// TIA Portal V20 export
FUNCTION "CallManualOperationLines_Unit1" : Void   // FC80, LAD
// stored: SetENOAutomatically false
   VAR_TEMP
      StatusEm : Array[0..13] of Struct
         Status : Array[0..40] of Word;
      END_STRUCT;
      errorIDEm : Array[0..13] of Struct
         errorID : Array[0..40] of Word;
      END_STRUCT;
      disableUnit1 : Bool;
      TempAxisCommands : "LBC_typeAxis64PosManualCommands";
      TempAxisMonitoring : "LBC_typeAxis64PosProcessValues";
      TempSoftCam : Array[0..8] of "LER_typeSoftCamParameter";
   END_VAR
   VAR CONSTANT
      MECHANIC_NAME_ENABLE : Bool;
   END_VAR
   VAR_TEMP   // added for the SCL form of the ladder/FBD networks
      _w1 : Bool;
   END_VAR
BEGIN

REGION Network 1: Unit 1 Enable Manual Operation
   // Condition to disable manual operation lines in Unit 3
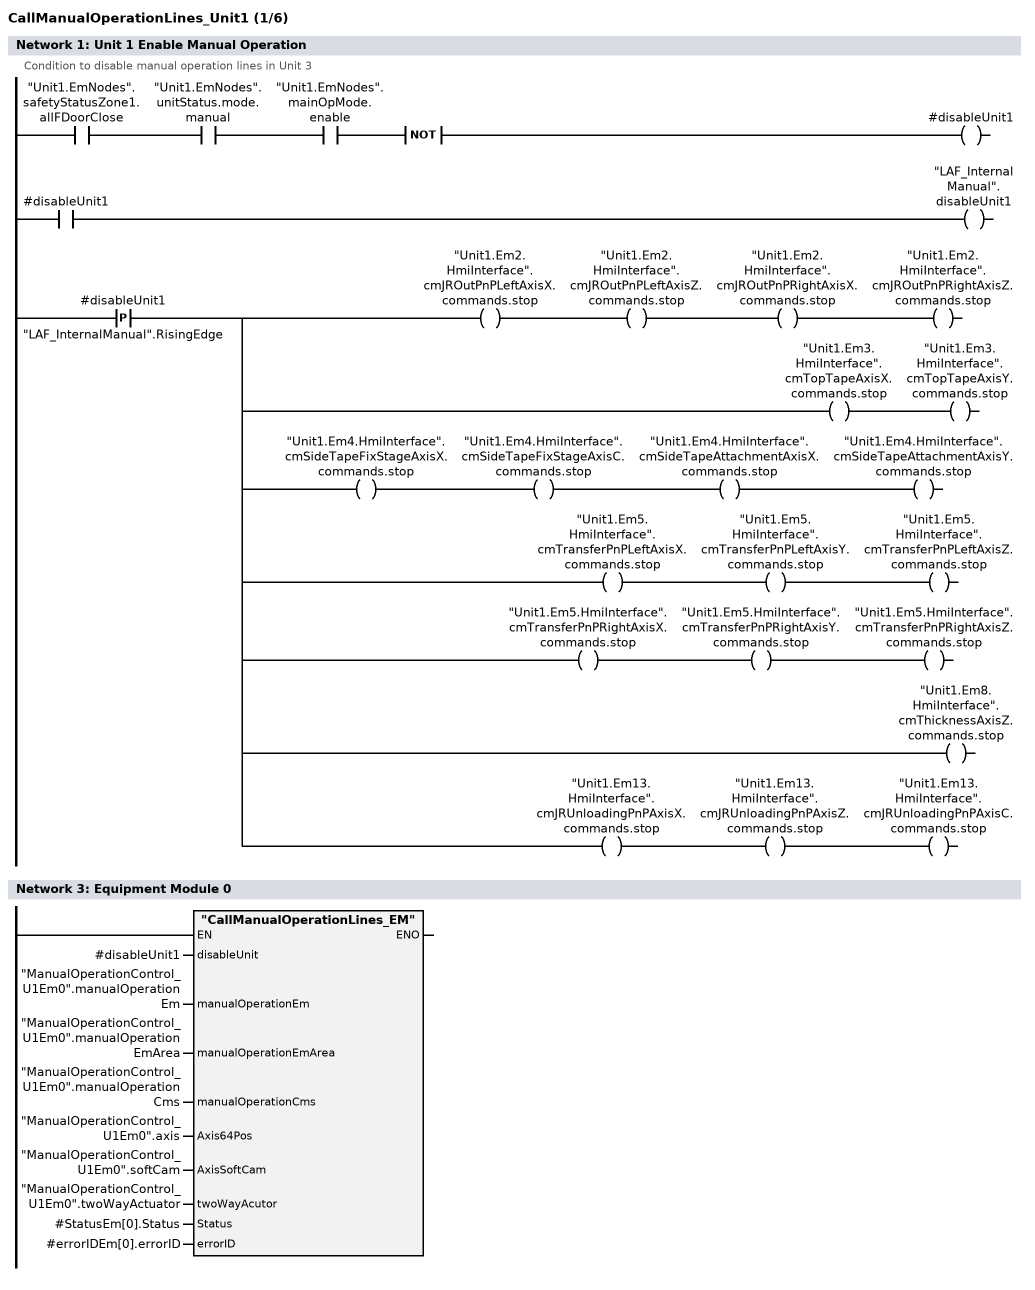
   RUNG wire#powerrail
      Contact( "Unit1.EmNodes".safetyStatusZone1.allFDoorClose )
      Contact( "Unit1.EmNodes".unitStatus.mode.manual )
      Contact( "Unit1.EmNodes".mainOpMode.enable )
      Not()
      Coil( #disableUnit1 )
   END_RUNG
   RUNG wire#powerrail
      Contact( #disableUnit1 )
      Coil( "LAF_InternalManual".disableUnit1 )
   END_RUNG
   RUNG wire#powerrail
      P_Contact(operand := #disableUnit1, bit := "LAF_InternalManual".RisingEdge)
      wire#w1
      Coil( "Unit1.Em2.HmiInterface".cmJROutPnPLeftAxisX.commands.stop )
      Coil( "Unit1.Em2.HmiInterface".cmJROutPnPLeftAxisZ.commands.stop )
      Coil( "Unit1.Em2.HmiInterface".cmJROutPnPRightAxisX.commands.stop )
      Coil( "Unit1.Em2.HmiInterface".cmJROutPnPRightAxisZ.commands.stop )
   END_RUNG
   RUNG wire#w1
      Coil( "Unit1.Em3.HmiInterface".cmTopTapeAxisX.commands.stop )
      Coil( "Unit1.Em3.HmiInterface".cmTopTapeAxisY.commands.stop )
   END_RUNG
   RUNG wire#w1
      Coil( "Unit1.Em4.HmiInterface".cmSideTapeFixStageAxisX.commands.stop )
      Coil( "Unit1.Em4.HmiInterface".cmSideTapeFixStageAxisC.commands.stop )
      Coil( "Unit1.Em4.HmiInterface".cmSideTapeAttachmentAxisX.commands.stop )
      Coil( "Unit1.Em4.HmiInterface".cmSideTapeAttachmentAxisY.commands.stop )
   END_RUNG
   RUNG wire#w1
      Coil( "Unit1.Em5.HmiInterface".cmTransferPnPLeftAxisX.commands.stop )
      Coil( "Unit1.Em5.HmiInterface".cmTransferPnPLeftAxisY.commands.stop )
      Coil( "Unit1.Em5.HmiInterface".cmTransferPnPLeftAxisZ.commands.stop )
   END_RUNG
   RUNG wire#w1
      Coil( "Unit1.Em5.HmiInterface".cmTransferPnPRightAxisX.commands.stop )
      Coil( "Unit1.Em5.HmiInterface".cmTransferPnPRightAxisY.commands.stop )
      Coil( "Unit1.Em5.HmiInterface".cmTransferPnPRightAxisZ.commands.stop )
   END_RUNG
   RUNG wire#w1
      Coil( "Unit1.Em8.HmiInterface".cmThicknessAxisZ.commands.stop )
   END_RUNG
   RUNG wire#w1
      Coil( "Unit1.Em13.HmiInterface".cmJRUnloadingPnPAxisX.commands.stop )
      Coil( "Unit1.Em13.HmiInterface".cmJRUnloadingPnPAxisZ.commands.stop )
      Coil( "Unit1.Em13.HmiInterface".cmJRUnloadingPnPAxisC.commands.stop )
   END_RUNG
   // the same network as SCL:
   #disableUnit1 := NOT ("Unit1.EmNodes".safetyStatusZone1.allFDoorClose AND "Unit1.EmNodes".unitStatus.mode.manual AND "Unit1.EmNodes".mainOpMode.enable);
   "LAF_InternalManual".disableUnit1 := #disableUnit1;
   #_w1 := #disableUnit1 AND NOT "LAF_InternalManual".RisingEdge;   // rising edge of #disableUnit1
   "LAF_InternalManual".RisingEdge := #disableUnit1;
   "Unit1.Em2.HmiInterface".cmJROutPnPLeftAxisX.commands.stop := #_w1;
   "Unit1.Em2.HmiInterface".cmJROutPnPLeftAxisZ.commands.stop := #_w1;
   "Unit1.Em2.HmiInterface".cmJROutPnPRightAxisX.commands.stop := #_w1;
   "Unit1.Em2.HmiInterface".cmJROutPnPRightAxisZ.commands.stop := #_w1;
   "Unit1.Em3.HmiInterface".cmTopTapeAxisX.commands.stop := #_w1;
   "Unit1.Em3.HmiInterface".cmTopTapeAxisY.commands.stop := #_w1;
   "Unit1.Em4.HmiInterface".cmSideTapeFixStageAxisX.commands.stop := #_w1;
   "Unit1.Em4.HmiInterface".cmSideTapeFixStageAxisC.commands.stop := #_w1;
   "Unit1.Em4.HmiInterface".cmSideTapeAttachmentAxisX.commands.stop := #_w1;
   "Unit1.Em4.HmiInterface".cmSideTapeAttachmentAxisY.commands.stop := #_w1;
   "Unit1.Em5.HmiInterface".cmTransferPnPLeftAxisX.commands.stop := #_w1;
   "Unit1.Em5.HmiInterface".cmTransferPnPLeftAxisY.commands.stop := #_w1;
   "Unit1.Em5.HmiInterface".cmTransferPnPLeftAxisZ.commands.stop := #_w1;
   "Unit1.Em5.HmiInterface".cmTransferPnPRightAxisX.commands.stop := #_w1;
   "Unit1.Em5.HmiInterface".cmTransferPnPRightAxisY.commands.stop := #_w1;
   "Unit1.Em5.HmiInterface".cmTransferPnPRightAxisZ.commands.stop := #_w1;
   "Unit1.Em8.HmiInterface".cmThicknessAxisZ.commands.stop := #_w1;
   "Unit1.Em13.HmiInterface".cmJRUnloadingPnPAxisX.commands.stop := #_w1;
   "Unit1.Em13.HmiInterface".cmJRUnloadingPnPAxisZ.commands.stop := #_w1;
   "Unit1.Em13.HmiInterface".cmJRUnloadingPnPAxisC.commands.stop := #_w1;
END_REGION

REGION Network 2 (SCL): Equipment Module 0 Cms Mapping
   REGION Input Mapping
       // TwoWayActuator
       "ManualOperationControl_U1Em0".twoWayActuator[1].monitoring := "Unit1.Em0.HmiInterface".cmStacker1NgBoxClampMoverOpenClose.monitoring;
       "ManualOperationControl_U1Em0".twoWayActuator[2].monitoring := "Unit1.Em0.HmiInterface".cmStacker1NgBoxClampLeftOpenClose.monitoring;
       "ManualOperationControl_U1Em0".twoWayActuator[3].monitoring := "Unit1.Em0.HmiInterface".cmStacker1NgBoxClampRightOpenClose.monitoring;
       "ManualOperationControl_U1Em0".twoWayActuator[4].monitoring := "Unit1.Em0.HmiInterface".cmStacker1NgBoxLoadingUpDown.monitoring;
       "ManualOperationControl_U1Em0".twoWayActuator[5].monitoring := "Unit1.Em0.HmiInterface".cmStacker1NgBoxUnitMoverBwdFwd.monitoring;
       "ManualOperationControl_U1Em0".twoWayActuator[6].monitoring := "Unit1.Em0.HmiInterface".cmStacker1NgBoxLiftDownUp.monitoring;
       "ManualOperationControl_U1Em0".twoWayActuator[7].monitoring := "Unit1.Em0.HmiInterface".cmStacker1NgBoxLockDownUp.monitoring;
   END_REGION


   REGION Output Mapping
       // TwoWayActuator
       "Unit1.Em0.HmiInterface".cmStacker1NgBoxClampMoverOpenClose.commands := "ManualOperationControl_U1Em0".twoWayActuator[1].commands;
       "Unit1.Em0.HmiInterface".cmStacker1NgBoxClampLeftOpenClose.commands := "ManualOperationControl_U1Em0".twoWayActuator[2].commands;
       "Unit1.Em0.HmiInterface".cmStacker1NgBoxClampRightOpenClose.commands := "ManualOperationControl_U1Em0".twoWayActuator[3].commands;
       "Unit1.Em0.HmiInterface".cmStacker1NgBoxLoadingUpDown.commands := "ManualOperationControl_U1Em0".twoWayActuator[4].commands;
       "Unit1.Em0.HmiInterface".cmStacker1NgBoxUnitMoverBwdFwd.commands := "ManualOperationControl_U1Em0".twoWayActuator[5].commands;
       "Unit1.Em0.HmiInterface".cmStacker1NgBoxLiftDownUp.commands := "ManualOperationControl_U1Em0".twoWayActuator[6].commands;
       "Unit1.Em0.HmiInterface".cmStacker1NgBoxLockDownUp.commands := "ManualOperationControl_U1Em0".twoWayActuator[7].commands;
   END_REGION
END_REGION

REGION Network 3: Equipment Module 0
   RUNG wire#powerrail
      "CallManualOperationLines_EM"(disableUnit := #disableUnit1, manualOperationEm := "ManualOperationControl_U1Em0".manualOperationEm, manualOperationEmArea := "ManualOperationControl_U1Em0".manualOperationEmArea, manualOperationCms := "ManualOperationControl_U1Em0".manualOperationCms, Axis64Pos := "ManualOperationControl_U1Em0".axis, AxisSoftCam := "ManualOperationControl_U1Em0".softCam, twoWayAcutor := "ManualOperationControl_U1Em0".twoWayActuator, Status := #StatusEm[0].Status, errorID := #errorIDEm[0].errorID)
   END_RUNG
   // the same network as SCL:
   "CallManualOperationLines_EM"(disableUnit := #disableUnit1,
                           manualOperationEm := "ManualOperationControl_U1Em0".manualOperationEm,
                           manualOperationEmArea := "ManualOperationControl_U1Em0".manualOperationEmArea,
                           manualOperationCms := "ManualOperationControl_U1Em0".manualOperationCms,
                           Axis64Pos := "ManualOperationControl_U1Em0".axis,
                           AxisSoftCam := "ManualOperationControl_U1Em0".softCam,
                           twoWayAcutor := "ManualOperationControl_U1Em0".twoWayActuator,
                           Status := #StatusEm[0].Status,
                           errorID := #errorIDEm[0].errorID);
END_REGION

REGION Network 4 (SCL): Equipment Module 1 Cms Mapping
   REGION Input Mapping
       // TwoWayActuator
       "ManualOperationControl_U1Em1".twoWayActuator[1].monitoring := "Unit1.Em1.HmiInterface".cmStacker2NgBoxClampMoverOpenClose.monitoring;
       "ManualOperationControl_U1Em1".twoWayActuator[2].monitoring := "Unit1.Em1.HmiInterface".cmStacker2NgBoxClampLeftOpenClose.monitoring;
       "ManualOperationControl_U1Em1".twoWayActuator[3].monitoring := "Unit1.Em1.HmiInterface".cmStacker2NgBoxClampRightOpenClose.monitoring;
       "ManualOperationControl_U1Em1".twoWayActuator[4].monitoring := "Unit1.Em1.HmiInterface".cmStacker2NgBoxLoadingUpDown.monitoring;
       "ManualOperationControl_U1Em1".twoWayActuator[5].monitoring := "Unit1.Em1.HmiInterface".cmStacker2NgBoxUnitMoverBwdFwd.monitoring;
       "ManualOperationControl_U1Em1".twoWayActuator[6].monitoring := "Unit1.Em1.HmiInterface".cmStacker2NgBoxLiftDownUp.monitoring;
       "ManualOperationControl_U1Em1".twoWayActuator[7].monitoring := "Unit1.Em1.HmiInterface".cmStacker2NgBoxLockDownUp.monitoring;
   END_REGION


   REGION Output Mapping  
       // TwoWayActuator
       "Unit1.Em1.HmiInterface".cmStacker2NgBoxClampMoverOpenClose.commands := "ManualOperationControl_U1Em1".twoWayActuator[1].commands;
       "Unit1.Em1.HmiInterface".cmStacker2NgBoxClampLeftOpenClose.commands := "ManualOperationControl_U1Em1".twoWayActuator[2].commands;
       "Unit1.Em1.HmiInterface".cmStacker2NgBoxClampRightOpenClose.commands := "ManualOperationControl_U1Em1".twoWayActuator[3].commands;
       "Unit1.Em1.HmiInterface".cmStacker2NgBoxLoadingUpDown.commands := "ManualOperationControl_U1Em1".twoWayActuator[4].commands;
       "Unit1.Em1.HmiInterface".cmStacker2NgBoxUnitMoverBwdFwd.commands := "ManualOperationControl_U1Em1".twoWayActuator[5].commands;
       "Unit1.Em1.HmiInterface".cmStacker2NgBoxLiftDownUp.commands := "ManualOperationControl_U1Em1".twoWayActuator[6].commands;
       "Unit1.Em1.HmiInterface".cmStacker2NgBoxLockDownUp.commands := "ManualOperationControl_U1Em1".twoWayActuator[7].commands;
   END_REGION
END_REGION

REGION Network 5: Equipment Module 1
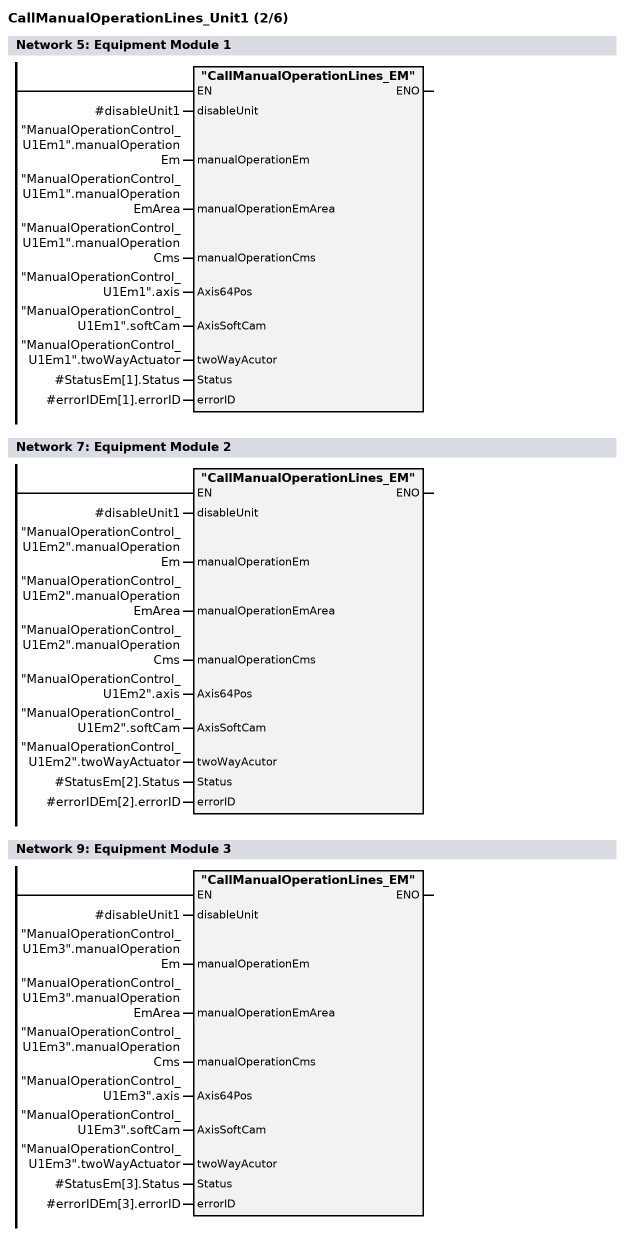
   RUNG wire#powerrail
      "CallManualOperationLines_EM"(disableUnit := #disableUnit1, manualOperationEm := "ManualOperationControl_U1Em1".manualOperationEm, manualOperationEmArea := "ManualOperationControl_U1Em1".manualOperationEmArea, manualOperationCms := "ManualOperationControl_U1Em1".manualOperationCms, Axis64Pos := "ManualOperationControl_U1Em1".axis, AxisSoftCam := "ManualOperationControl_U1Em1".softCam, twoWayAcutor := "ManualOperationControl_U1Em1".twoWayActuator, Status := #StatusEm[1].Status, errorID := #errorIDEm[1].errorID)
   END_RUNG
   // the same network as SCL:
   "CallManualOperationLines_EM"(disableUnit := #disableUnit1,
                           manualOperationEm := "ManualOperationControl_U1Em1".manualOperationEm,
                           manualOperationEmArea := "ManualOperationControl_U1Em1".manualOperationEmArea,
                           manualOperationCms := "ManualOperationControl_U1Em1".manualOperationCms,
                           Axis64Pos := "ManualOperationControl_U1Em1".axis,
                           AxisSoftCam := "ManualOperationControl_U1Em1".softCam,
                           twoWayAcutor := "ManualOperationControl_U1Em1".twoWayActuator,
                           Status := #StatusEm[1].Status,
                           errorID := #errorIDEm[1].errorID);
END_REGION

REGION Network 6 (SCL): Equipment Module 2 Cms Mapping
   REGION Input Mapping
       // Axis
       "ManualOperationControl_U1Em2".axis[1].monitoring := "Unit1.Em2.HmiInterface".cmJROutPnPLeftAxisX.monitoring;
       "ManualOperationControl_U1Em2".axis[2].monitoring := "Unit1.Em2.HmiInterface".cmJROutPnPLeftAxisZ.monitoring;
       "ManualOperationControl_U1Em2".axis[3].monitoring := "Unit1.Em2.HmiInterface".cmJROutPnPRightAxisX.monitoring;
       "ManualOperationControl_U1Em2".axis[4].monitoring := "Unit1.Em2.HmiInterface".cmJROutPnPRightAxisZ.monitoring;

       // SoftCam
       "ManualOperationControl_U1Em2".softCam[1] := "Unit1.Em2.HmiInterface".cm.softcam.jrOutPnPLeftAxisX;
       "ManualOperationControl_U1Em2".softCam[2] := "Unit1.Em2.HmiInterface".cm.softcam.jrOutPnPLeftAxisZ;
       "ManualOperationControl_U1Em2".softCam[3] := "Unit1.Em2.HmiInterface".cm.softcam.jrOutPnPRightAxisX;
       "ManualOperationControl_U1Em2".softCam[4] := "Unit1.Em2.HmiInterface".cm.softcam.jrOutPnPRightAxisZ;

       // TwoWayActuator
       "ManualOperationControl_U1Em2".twoWayActuator[1].monitoring := "Unit1.Em2.HmiInterface".cmJROutPnPLeftClampOpenClose.monitoring;
       "ManualOperationControl_U1Em2".twoWayActuator[2].monitoring := "Unit1.Em2.HmiInterface".cmJROutPnPRightClampOpenClose.monitoring;
   END_REGION


   REGION Output Mapping
       // Axis
       "Unit1.Em2.HmiInterface".cmJROutPnPLeftAxisX.commands.jogForward := "ManualOperationControl_U1Em2".axis[1].commands.jogForward;
       "Unit1.Em2.HmiInterface".cmJROutPnPLeftAxisX.commands.jogBackward := "ManualOperationControl_U1Em2".axis[1].commands.jogBackward;
       "Unit1.Em2.HmiInterface".cmJROutPnPLeftAxisZ.commands.jogForward := "ManualOperationControl_U1Em2".axis[2].commands.jogForward;
       "Unit1.Em2.HmiInterface".cmJROutPnPLeftAxisZ.commands.jogBackward := "ManualOperationControl_U1Em2".axis[2].commands.jogBackward;
       "Unit1.Em2.HmiInterface".cmJROutPnPRightAxisX.commands.jogForward := "ManualOperationControl_U1Em2".axis[3].commands.jogForward;
       "Unit1.Em2.HmiInterface".cmJROutPnPRightAxisX.commands.jogBackward := "ManualOperationControl_U1Em2".axis[3].commands.jogBackward;
       "Unit1.Em2.HmiInterface".cmJROutPnPRightAxisZ.commands.jogForward := "ManualOperationControl_U1Em2".axis[4].commands.jogForward;
       "Unit1.Em2.HmiInterface".cmJROutPnPRightAxisZ.commands.jogBackward := "ManualOperationControl_U1Em2".axis[4].commands.jogBackward;

       // TwoWayActuator
       "Unit1.Em2.HmiInterface".cmJROutPnPLeftClampOpenClose.commands := "ManualOperationControl_U1Em2".twoWayActuator[1].commands;
       "Unit1.Em2.HmiInterface".cmJROutPnPRightClampOpenClose.commands := "ManualOperationControl_U1Em2".twoWayActuator[2].commands;
   END_REGION
END_REGION

REGION Network 7: Equipment Module 2
   RUNG wire#powerrail
      "CallManualOperationLines_EM"(disableUnit := #disableUnit1, manualOperationEm := "ManualOperationControl_U1Em2".manualOperationEm, manualOperationEmArea := "ManualOperationControl_U1Em2".manualOperationEmArea, manualOperationCms := "ManualOperationControl_U1Em2".manualOperationCms, Axis64Pos := "ManualOperationControl_U1Em2".axis, AxisSoftCam := "ManualOperationControl_U1Em2".softCam, twoWayAcutor := "ManualOperationControl_U1Em2".twoWayActuator, Status := #StatusEm[2].Status, errorID := #errorIDEm[2].errorID)
   END_RUNG
   // the same network as SCL:
   "CallManualOperationLines_EM"(disableUnit := #disableUnit1,
                           manualOperationEm := "ManualOperationControl_U1Em2".manualOperationEm,
                           manualOperationEmArea := "ManualOperationControl_U1Em2".manualOperationEmArea,
                           manualOperationCms := "ManualOperationControl_U1Em2".manualOperationCms,
                           Axis64Pos := "ManualOperationControl_U1Em2".axis,
                           AxisSoftCam := "ManualOperationControl_U1Em2".softCam,
                           twoWayAcutor := "ManualOperationControl_U1Em2".twoWayActuator,
                           Status := #StatusEm[2].Status,
                           errorID := #errorIDEm[2].errorID);
END_REGION

REGION Network 8 (SCL): Equipment Module 3 Cms Mapping
   REGION Input Mapping
        // Axis
       "ManualOperationControl_U1Em3".axis[1].monitoring := "Unit1.Em3.HmiInterface".cmTopTapeAxisX.monitoring;
       "ManualOperationControl_U1Em3".axis[2].monitoring := "Unit1.Em3.HmiInterface".cmTopTapeAxisY.monitoring;

       // SoftCam
       "ManualOperationControl_U1Em3".softCam[1] := "Unit1.Em3.HmiInterface".cm.softcam.topTapeAxisX;
       "ManualOperationControl_U1Em3".softCam[2] := "Unit1.Em3.HmiInterface".cm.softcam.topTapeAxisY;

       // TwoWayActuator
       "ManualOperationControl_U1Em3".twoWayActuator[1].monitoring := "Unit1.Em3.HmiInterface".cmTopTapeCutterUpDown.monitoring;
       "ManualOperationControl_U1Em3".twoWayActuator[2].monitoring := "Unit1.Em3.HmiInterface".cmTopTapeCutterClampUpDown.monitoring;
       "ManualOperationControl_U1Em3".twoWayActuator[3].monitoring := "Unit1.Em3.HmiInterface".cmTopTapeLoadingClampOpenClose.monitoring;
       "ManualOperationControl_U1Em3".twoWayActuator[4].monitoring := "Unit1.Em3.HmiInterface".cmTopTapeTensionBwdFwd.monitoring;
       "ManualOperationControl_U1Em3".twoWayActuator[5].monitoring := "Unit1.Em3.HmiInterface".cmTopTapeLoadingBwdFwd.monitoring;
       "ManualOperationControl_U1Em3".twoWayActuator[6].monitoring := "Unit1.Em3.HmiInterface".cmTopTapeClampTopLeftUpDown.monitoring;
       "ManualOperationControl_U1Em3".twoWayActuator[7].monitoring := "Unit1.Em3.HmiInterface".cmTopTapeClampTopCenterUpDown.monitoring;
       "ManualOperationControl_U1Em3".twoWayActuator[8].monitoring := "Unit1.Em3.HmiInterface".cmTopTapeClampTopRightUpDown.monitoring;
       "ManualOperationControl_U1Em3".twoWayActuator[9].monitoring := "Unit1.Em3.HmiInterface".cmTopTapeClampBtmDownUp.monitoring;
       "ManualOperationControl_U1Em3".twoWayActuator[10].monitoring := "Unit1.Em3.HmiInterface".cmTopTapeAttachmentUpDown.monitoring;
       "ManualOperationControl_U1Em3".twoWayActuator[11].monitoring := "Unit1.Em3.HmiInterface".cmTopTapeAttachmentVaccumOffOn.monitoring;

   END_REGION


   REGION Output Mapping
       // Axis
       "Unit1.Em3.HmiInterface".cmTopTapeAxisX.commands.jogForward := "ManualOperationControl_U1Em3".axis[1].commands.jogForward;
       "Unit1.Em3.HmiInterface".cmTopTapeAxisX.commands.jogBackward := "ManualOperationControl_U1Em3".axis[1].commands.jogBackward;
       "Unit1.Em3.HmiInterface".cmTopTapeAxisY.commands.jogForward := "ManualOperationControl_U1Em3".axis[2].commands.jogForward;
       "Unit1.Em3.HmiInterface".cmTopTapeAxisY.commands.jogBackward := "ManualOperationControl_U1Em3".axis[2].commands.jogBackward;

       // TwoWayActuator
       "Unit1.Em3.HmiInterface".cmTopTapeCutterUpDown.commands := "ManualOperationControl_U1Em3".twoWayActuator[1].commands;
       "Unit1.Em3.HmiInterface".cmTopTapeCutterClampUpDown.commands := "ManualOperationControl_U1Em3".twoWayActuator[2].commands;
       "Unit1.Em3.HmiInterface".cmTopTapeLoadingClampOpenClose.commands := "ManualOperationControl_U1Em3".twoWayActuator[3].commands;
       "Unit1.Em3.HmiInterface".cmTopTapeTensionBwdFwd.commands := "ManualOperationControl_U1Em3".twoWayActuator[4].commands;
       "Unit1.Em3.HmiInterface".cmTopTapeLoadingBwdFwd.commands := "ManualOperationControl_U1Em3".twoWayActuator[5].commands;
       "Unit1.Em3.HmiInterface".cmTopTapeClampTopLeftUpDown.commands := "ManualOperationControl_U1Em3".twoWayActuator[6].commands;
       "Unit1.Em3.HmiInterface".cmTopTapeClampTopCenterUpDown.commands := "ManualOperationControl_U1Em3".twoWayActuator[7].commands;
       "Unit1.Em3.HmiInterface".cmTopTapeClampTopRightUpDown.commands := "ManualOperationControl_U1Em3".twoWayActuator[8].commands;
       "Unit1.Em3.HmiInterface".cmTopTapeClampBtmDownUp.commands := "ManualOperationControl_U1Em3".twoWayActuator[9].commands;
       "Unit1.Em3.HmiInterface".cmTopTapeAttachmentUpDown.commands := "ManualOperationControl_U1Em3".twoWayActuator[10].commands;
       "Unit1.Em3.HmiInterface".cmTopTapeAttachmentVaccumOffOn.commands := "ManualOperationControl_U1Em3".twoWayActuator[11].commands;

   END_REGION
END_REGION

REGION Network 9: Equipment Module 3
   RUNG wire#powerrail
      "CallManualOperationLines_EM"(disableUnit := #disableUnit1, manualOperationEm := "ManualOperationControl_U1Em3".manualOperationEm, manualOperationEmArea := "ManualOperationControl_U1Em3".manualOperationEmArea, manualOperationCms := "ManualOperationControl_U1Em3".manualOperationCms, Axis64Pos := "ManualOperationControl_U1Em3".axis, AxisSoftCam := "ManualOperationControl_U1Em3".softCam, twoWayAcutor := "ManualOperationControl_U1Em3".twoWayActuator, Status := #StatusEm[3].Status, errorID := #errorIDEm[3].errorID)
   END_RUNG
   // the same network as SCL:
   "CallManualOperationLines_EM"(disableUnit := #disableUnit1,
                           manualOperationEm := "ManualOperationControl_U1Em3".manualOperationEm,
                           manualOperationEmArea := "ManualOperationControl_U1Em3".manualOperationEmArea,
                           manualOperationCms := "ManualOperationControl_U1Em3".manualOperationCms,
                           Axis64Pos := "ManualOperationControl_U1Em3".axis,
                           AxisSoftCam := "ManualOperationControl_U1Em3".softCam,
                           twoWayAcutor := "ManualOperationControl_U1Em3".twoWayActuator,
                           Status := #StatusEm[3].Status,
                           errorID := #errorIDEm[3].errorID);
END_REGION

REGION Network 10 (SCL): Equipment Module 4 Cms Mapping
   REGION Input Mapping
       // Axis
       "ManualOperationControl_U1Em4".axis[1].monitoring := "Unit1.Em4.HmiInterface".cmSideTapeFixStageAxisX.monitoring;
       "ManualOperationControl_U1Em4".axis[2].monitoring := "Unit1.Em4.HmiInterface".cmSideTapeFixStageAxisC.monitoring;
       "ManualOperationControl_U1Em4".axis[3].monitoring := "Unit1.Em4.HmiInterface".cmSideTapeAttachmentAxisX.monitoring;
       "ManualOperationControl_U1Em4".axis[4].monitoring := "Unit1.Em4.HmiInterface".cmSideTapeAttachmentAxisY.monitoring;

       // SoftCam
       "ManualOperationControl_U1Em4".softCam[1] := "Unit1.Em4.HmiInterface".cm.softcam.sideTapeFixStageAxisX;
       "ManualOperationControl_U1Em4".softCam[2] := "Unit1.Em4.HmiInterface".cm.softcam.sideTapeFixStageAxisC;
       "ManualOperationControl_U1Em4".softCam[3] := "Unit1.Em4.HmiInterface".cm.softcam.sideTapeAttachmentAxisX;
       "ManualOperationControl_U1Em4".softCam[4] := "Unit1.Em4.HmiInterface".cm.softcam.sideTapeAttachmentAxisY;

       // TwoWayActuator
       "ManualOperationControl_U1Em4".twoWayActuator[1].monitoring := "Unit1.Em4.HmiInterface".cmSideTapeCutterBwdFwd.monitoring;
       "ManualOperationControl_U1Em4".twoWayActuator[2].monitoring := "Unit1.Em4.HmiInterface".cmSideTapeCutterClampBwdFwd.monitoring;
       "ManualOperationControl_U1Em4".twoWayActuator[3].monitoring := "Unit1.Em4.HmiInterface".cmSideTapeLoadingClampOpenClose.monitoring;
       "ManualOperationControl_U1Em4".twoWayActuator[4].monitoring := "Unit1.Em4.HmiInterface".cmSideTapeLoadingDownUp.monitoring;
       "ManualOperationControl_U1Em4".twoWayActuator[5].monitoring := "Unit1.Em4.HmiInterface".cmSideTapeTensionBwdFwd.monitoring;
       "ManualOperationControl_U1Em4".twoWayActuator[6].monitoring := "Unit1.Em4.HmiInterface".cmSideTapeAttachmentLeftBwdFwd.monitoring;
       "ManualOperationControl_U1Em4".twoWayActuator[7].monitoring := "Unit1.Em4.HmiInterface".cmSideTapeAttachmentRightBwdFwd.monitoring;
       "ManualOperationControl_U1Em4".twoWayActuator[8].monitoring := "Unit1.Em4.HmiInterface".cmSideTapeAttachmentBtmBwdFwd.monitoring;
       "ManualOperationControl_U1Em4".twoWayActuator[9].monitoring := "Unit1.Em4.HmiInterface".cmSideTapeFixStageClampOpenClose.monitoring;
       "ManualOperationControl_U1Em4".twoWayActuator[10].monitoring := "Unit1.Em4.HmiInterface".cmSideTapeAttachment1TopVaccumOffOn.monitoring;
       "ManualOperationControl_U1Em4".twoWayActuator[11].monitoring := "Unit1.Em4.HmiInterface".cmSideTapeAttachment1BtmVaccumOffOn.monitoring;
       "ManualOperationControl_U1Em4".twoWayActuator[12].monitoring := "Unit1.Em4.HmiInterface".cmSideTapeAttachment2TopVaccumOffOn.monitoring;
       "ManualOperationControl_U1Em4".twoWayActuator[13].monitoring := "Unit1.Em4.HmiInterface".cmSideTapeAttachment2BtmVaccumOffOn.monitoring;

   END_REGION


   REGION Output Mapping
       // Axis
       "Unit1.Em4.HmiInterface".cmSideTapeFixStageAxisX.commands.jogForward := "ManualOperationControl_U1Em4".axis[1].commands.jogForward;
       "Unit1.Em4.HmiInterface".cmSideTapeFixStageAxisX.commands.jogBackward := "ManualOperationControl_U1Em4".axis[1].commands.jogBackward;
       "Unit1.Em4.HmiInterface".cmSideTapeFixStageAxisC.commands.jogForward := "ManualOperationControl_U1Em4".axis[2].commands.jogForward;
       "Unit1.Em4.HmiInterface".cmSideTapeFixStageAxisC.commands.jogBackward := "ManualOperationControl_U1Em4".axis[2].commands.jogBackward;
       "Unit1.Em4.HmiInterface".cmSideTapeAttachmentAxisX.commands.jogForward := "ManualOperationControl_U1Em4".axis[3].commands.jogForward;
       "Unit1.Em4.HmiInterface".cmSideTapeAttachmentAxisX.commands.jogBackward := "ManualOperationControl_U1Em4".axis[3].commands.jogBackward;
       "Unit1.Em4.HmiInterface".cmSideTapeAttachmentAxisY.commands.jogForward := "ManualOperationControl_U1Em4".axis[4].commands.jogForward;
       "Unit1.Em4.HmiInterface".cmSideTapeAttachmentAxisY.commands.jogBackward := "ManualOperationControl_U1Em4".axis[4].commands.jogBackward;

       // TwoWayActuator
       "Unit1.Em4.HmiInterface".cmSideTapeCutterBwdFwd.commands := "ManualOperationControl_U1Em4".twoWayActuator[1].commands;
       "Unit1.Em4.HmiInterface".cmSideTapeCutterClampBwdFwd.commands := "ManualOperationControl_U1Em4".twoWayActuator[2].commands;
       "Unit1.Em4.HmiInterface".cmSideTapeLoadingClampOpenClose.commands := "ManualOperationControl_U1Em4".twoWayActuator[3].commands;
       "Unit1.Em4.HmiInterface".cmSideTapeLoadingDownUp.commands:= "ManualOperationControl_U1Em4".twoWayActuator[4].commands;
       "Unit1.Em4.HmiInterface".cmSideTapeTensionBwdFwd.commands := "ManualOperationControl_U1Em4".twoWayActuator[5].commands;
       "Unit1.Em4.HmiInterface".cmSideTapeAttachmentLeftBwdFwd.commands := "ManualOperationControl_U1Em4".twoWayActuator[6].commands;
       "Unit1.Em4.HmiInterface".cmSideTapeAttachmentRightBwdFwd.commands := "ManualOperationControl_U1Em4".twoWayActuator[7].commands;
       "Unit1.Em4.HmiInterface".cmSideTapeAttachmentBtmBwdFwd.commands := "ManualOperationControl_U1Em4".twoWayActuator[8].commands;
       "Unit1.Em4.HmiInterface".cmSideTapeFixStageClampOpenClose.commands := "ManualOperationControl_U1Em4".twoWayActuator[9].commands;
       "Unit1.Em4.HmiInterface".cmSideTapeAttachment1TopVaccumOffOn.commands := "ManualOperationControl_U1Em4".twoWayActuator[10].commands;
       "Unit1.Em4.HmiInterface".cmSideTapeAttachment1BtmVaccumOffOn.commands := "ManualOperationControl_U1Em4".twoWayActuator[11].commands;
       "Unit1.Em4.HmiInterface".cmSideTapeAttachment2TopVaccumOffOn.commands := "ManualOperationControl_U1Em4".twoWayActuator[12].commands;
       "Unit1.Em4.HmiInterface".cmSideTapeAttachment2BtmVaccumOffOn.commands := "ManualOperationControl_U1Em4".twoWayActuator[13].commands;

   END_REGION
END_REGION

REGION Network 11: Equipment Module 4
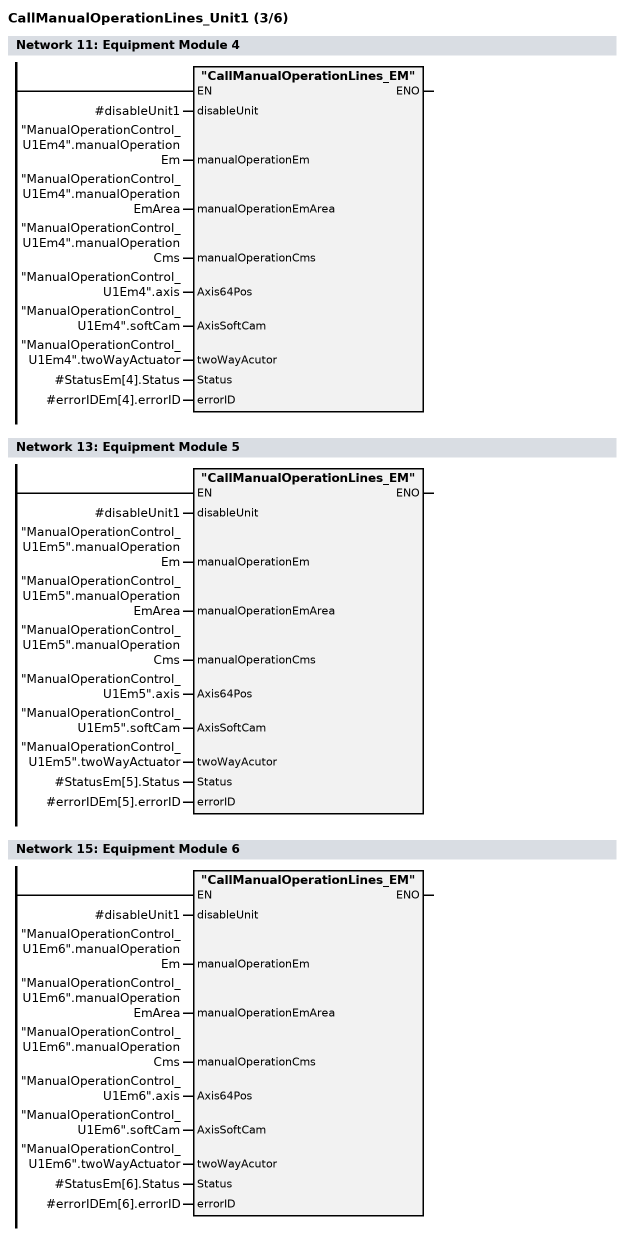
   RUNG wire#powerrail
      "CallManualOperationLines_EM"(disableUnit := #disableUnit1, manualOperationEm := "ManualOperationControl_U1Em4".manualOperationEm, manualOperationEmArea := "ManualOperationControl_U1Em4".manualOperationEmArea, manualOperationCms := "ManualOperationControl_U1Em4".manualOperationCms, Axis64Pos := "ManualOperationControl_U1Em4".axis, AxisSoftCam := "ManualOperationControl_U1Em4".softCam, twoWayAcutor := "ManualOperationControl_U1Em4".twoWayActuator, Status := #StatusEm[4].Status, errorID := #errorIDEm[4].errorID)
   END_RUNG
   // the same network as SCL:
   "CallManualOperationLines_EM"(disableUnit := #disableUnit1,
                           manualOperationEm := "ManualOperationControl_U1Em4".manualOperationEm,
                           manualOperationEmArea := "ManualOperationControl_U1Em4".manualOperationEmArea,
                           manualOperationCms := "ManualOperationControl_U1Em4".manualOperationCms,
                           Axis64Pos := "ManualOperationControl_U1Em4".axis,
                           AxisSoftCam := "ManualOperationControl_U1Em4".softCam,
                           twoWayAcutor := "ManualOperationControl_U1Em4".twoWayActuator,
                           Status := #StatusEm[4].Status,
                           errorID := #errorIDEm[4].errorID);
END_REGION

REGION Network 12 (SCL): Equipment Module 5 Cms Mapping
   REGION Input Mapping
        // Axis
       "ManualOperationControl_U1Em5".axis[1].monitoring := "Unit1.Em5.HmiInterface".cmTransferPnPLeftAxisX.monitoring;
       "ManualOperationControl_U1Em5".axis[2].monitoring := "Unit1.Em5.HmiInterface".cmTransferPnPLeftAxisY.monitoring;
       "ManualOperationControl_U1Em5".axis[3].monitoring := "Unit1.Em5.HmiInterface".cmTransferPnPLeftAxisZ.monitoring;
       "ManualOperationControl_U1Em5".axis[4].monitoring := "Unit1.Em5.HmiInterface".cmTransferPnPRightAxisX.monitoring;
       "ManualOperationControl_U1Em5".axis[5].monitoring := "Unit1.Em5.HmiInterface".cmTransferPnPRightAxisY.monitoring;
       "ManualOperationControl_U1Em5".axis[6].monitoring := "Unit1.Em5.HmiInterface".cmTransferPnPRightAxisZ.monitoring;

       // SoftCam
       "ManualOperationControl_U1Em5".softCam[1] := "Unit1.Em5.HmiInterface".cm.softcam.transferPnPLeftAxisX;
       "ManualOperationControl_U1Em5".softCam[2] := "Unit1.Em5.HmiInterface".cm.softcam.transferPnPLeftAxisY;
       "ManualOperationControl_U1Em5".softCam[3] := "Unit1.Em5.HmiInterface".cm.softcam.transferPnPLeftAxisZ;
       "ManualOperationControl_U1Em5".softCam[4] := "Unit1.Em5.HmiInterface".cm.softcam.transferPnPRightAxisX;
       "ManualOperationControl_U1Em5".softCam[5] := "Unit1.Em5.HmiInterface".cm.softcam.transferPnPRightAxisY;
       "ManualOperationControl_U1Em5".softCam[6] := "Unit1.Em5.HmiInterface".cm.softcam.transferPnPRightAxisZ;

       // TwoWayActuator
       "ManualOperationControl_U1Em5".twoWayActuator[1].monitoring := "Unit1.Em5.HmiInterface".cmTransferPnPLeftClampOpenClose.monitoring;
       "ManualOperationControl_U1Em5".twoWayActuator[2].monitoring := "Unit1.Em5.HmiInterface".cmTransferPnPRightClampOpenClose.monitoring;
   END_REGION


   REGION Output Mapping
       // Axis
       "Unit1.Em5.HmiInterface".cmTransferPnPLeftAxisX.commands.jogForward := "ManualOperationControl_U1Em5".axis[1].commands.jogForward;
       "Unit1.Em5.HmiInterface".cmTransferPnPLeftAxisX.commands.jogBackward := "ManualOperationControl_U1Em5".axis[1].commands.jogBackward;
       "Unit1.Em5.HmiInterface".cmTransferPnPLeftAxisY.commands.jogForward := "ManualOperationControl_U1Em5".axis[2].commands.jogForward;
       "Unit1.Em5.HmiInterface".cmTransferPnPLeftAxisY.commands.jogBackward := "ManualOperationControl_U1Em5".axis[2].commands.jogBackward;
       "Unit1.Em5.HmiInterface".cmTransferPnPLeftAxisZ.commands.jogForward := "ManualOperationControl_U1Em5".axis[3].commands.jogForward;
       "Unit1.Em5.HmiInterface".cmTransferPnPLeftAxisZ.commands.jogBackward := "ManualOperationControl_U1Em5".axis[3].commands.jogBackward;
       "Unit1.Em5.HmiInterface".cmTransferPnPRightAxisX.commands.jogForward := "ManualOperationControl_U1Em5".axis[4].commands.jogForward;
       "Unit1.Em5.HmiInterface".cmTransferPnPRightAxisX.commands.jogBackward := "ManualOperationControl_U1Em5".axis[4].commands.jogBackward;
       "Unit1.Em5.HmiInterface".cmTransferPnPRightAxisY.commands.jogForward := "ManualOperationControl_U1Em5".axis[5].commands.jogForward;
       "Unit1.Em5.HmiInterface".cmTransferPnPRightAxisY.commands.jogBackward := "ManualOperationControl_U1Em5".axis[5].commands.jogBackward;
       "Unit1.Em5.HmiInterface".cmTransferPnPRightAxisZ.commands.jogForward := "ManualOperationControl_U1Em5".axis[6].commands.jogForward;
       "Unit1.Em5.HmiInterface".cmTransferPnPRightAxisZ.commands.jogBackward := "ManualOperationControl_U1Em5".axis[6].commands.jogBackward;

       // TwoWayActuator
       "Unit1.Em5.HmiInterface".cmTransferPnPLeftClampOpenClose.commands := "ManualOperationControl_U1Em5".twoWayActuator[1].commands;
       "Unit1.Em5.HmiInterface".cmTransferPnPRightClampOpenClose.commands := "ManualOperationControl_U1Em5".twoWayActuator[2].commands;
   END_REGION
END_REGION

REGION Network 13: Equipment Module 5
   RUNG wire#powerrail
      "CallManualOperationLines_EM"(disableUnit := #disableUnit1, manualOperationEm := "ManualOperationControl_U1Em5".manualOperationEm, manualOperationEmArea := "ManualOperationControl_U1Em5".manualOperationEmArea, manualOperationCms := "ManualOperationControl_U1Em5".manualOperationCms, Axis64Pos := "ManualOperationControl_U1Em5".axis, AxisSoftCam := "ManualOperationControl_U1Em5".softCam, twoWayAcutor := "ManualOperationControl_U1Em5".twoWayActuator, Status := #StatusEm[5].Status, errorID := #errorIDEm[5].errorID)
   END_RUNG
   // the same network as SCL:
   "CallManualOperationLines_EM"(disableUnit := #disableUnit1,
                           manualOperationEm := "ManualOperationControl_U1Em5".manualOperationEm,
                           manualOperationEmArea := "ManualOperationControl_U1Em5".manualOperationEmArea,
                           manualOperationCms := "ManualOperationControl_U1Em5".manualOperationCms,
                           Axis64Pos := "ManualOperationControl_U1Em5".axis,
                           AxisSoftCam := "ManualOperationControl_U1Em5".softCam,
                           twoWayAcutor := "ManualOperationControl_U1Em5".twoWayActuator,
                           Status := #StatusEm[5].Status,
                           errorID := #errorIDEm[5].errorID);
END_REGION

REGION Network 14 (SCL): Equipment Module 6 Cms Mapping
   REGION Input Mapping  
       // TwoWayActuator
       "ManualOperationControl_U1Em6".twoWayActuator[3].monitoring := "Unit1.Em6.HmiInterface".cmHotpressLeftStageLiftFrontUpDown.monitoring;
       "ManualOperationControl_U1Em6".twoWayActuator[4].monitoring := "Unit1.Em6.HmiInterface".cmHotpressLeftStageLiftRearUpDown.monitoring;
   END_REGION


   REGION Output Mapping
       // TwoWayActuator
       "Unit1.Em6.HmiInterface".cmHotpressLeftStageLiftFrontUpDown.commands := "ManualOperationControl_U1Em6".twoWayActuator[3].commands;
       "Unit1.Em6.HmiInterface".cmHotpressLeftStageLiftRearUpDown.commands := "ManualOperationControl_U1Em6".twoWayActuator[4].commands;
   END_REGION
END_REGION

REGION Network 15: Equipment Module 6
   RUNG wire#powerrail
      "CallManualOperationLines_EM"(disableUnit := #disableUnit1, manualOperationEm := "ManualOperationControl_U1Em6".manualOperationEm, manualOperationEmArea := "ManualOperationControl_U1Em6".manualOperationEmArea, manualOperationCms := "ManualOperationControl_U1Em6".manualOperationCms, Axis64Pos := "ManualOperationControl_U1Em6".axis, AxisSoftCam := "ManualOperationControl_U1Em6".softCam, twoWayAcutor := "ManualOperationControl_U1Em6".twoWayActuator, Status := #StatusEm[6].Status, errorID := #errorIDEm[6].errorID)
   END_RUNG
   // the same network as SCL:
   "CallManualOperationLines_EM"(disableUnit := #disableUnit1,
                           manualOperationEm := "ManualOperationControl_U1Em6".manualOperationEm,
                           manualOperationEmArea := "ManualOperationControl_U1Em6".manualOperationEmArea,
                           manualOperationCms := "ManualOperationControl_U1Em6".manualOperationCms,
                           Axis64Pos := "ManualOperationControl_U1Em6".axis,
                           AxisSoftCam := "ManualOperationControl_U1Em6".softCam,
                           twoWayAcutor := "ManualOperationControl_U1Em6".twoWayActuator,
                           Status := #StatusEm[6].Status,
                           errorID := #errorIDEm[6].errorID);
END_REGION

REGION Network 16 (SCL): Equipment Module 7 Cms Mapping
   REGION Input Mapping  
       // TwoWayActuator
       "ManualOperationControl_U1Em7".twoWayActuator[3].monitoring := "Unit1.Em7.HmiInterface".cmHotPressRightStageLiftFrontUpDown.monitoring;
       "ManualOperationControl_U1Em7".twoWayActuator[4].monitoring := "Unit1.Em7.HmiInterface".cmHotPressRightStageLiftRearUpDown.monitoring;
   END_REGION


   REGION Output Mapping
       // TwoWayActuator
       "Unit1.Em7.HmiInterface".cmHotPressRightStageLiftFrontUpDown.commands := "ManualOperationControl_U1Em7".twoWayActuator[3].commands;
       "Unit1.Em7.HmiInterface".cmHotPressRightStageLiftRearUpDown.commands := "ManualOperationControl_U1Em7".twoWayActuator[4].commands;
   END_REGION
END_REGION

REGION Network 17: Equipment Module 7
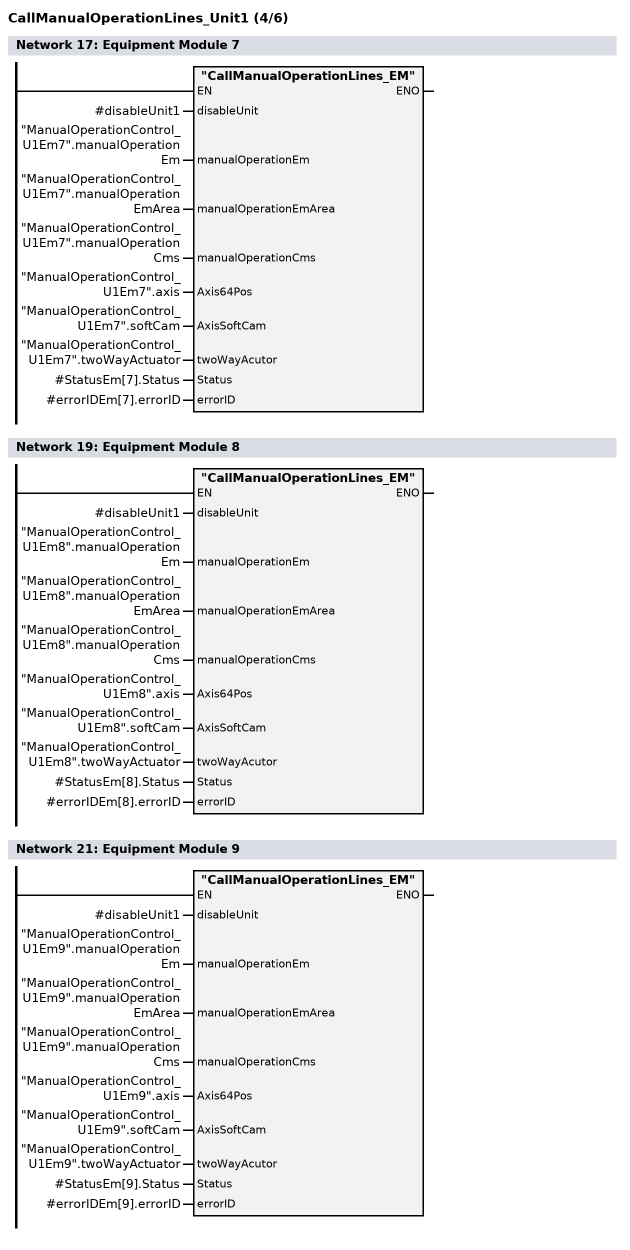
   RUNG wire#powerrail
      "CallManualOperationLines_EM"(disableUnit := #disableUnit1, manualOperationEm := "ManualOperationControl_U1Em7".manualOperationEm, manualOperationEmArea := "ManualOperationControl_U1Em7".manualOperationEmArea, manualOperationCms := "ManualOperationControl_U1Em7".manualOperationCms, Axis64Pos := "ManualOperationControl_U1Em7".axis, AxisSoftCam := "ManualOperationControl_U1Em7".softCam, twoWayAcutor := "ManualOperationControl_U1Em7".twoWayActuator, Status := #StatusEm[7].Status, errorID := #errorIDEm[7].errorID)
   END_RUNG
   // the same network as SCL:
   "CallManualOperationLines_EM"(disableUnit := #disableUnit1,
                           manualOperationEm := "ManualOperationControl_U1Em7".manualOperationEm,
                           manualOperationEmArea := "ManualOperationControl_U1Em7".manualOperationEmArea,
                           manualOperationCms := "ManualOperationControl_U1Em7".manualOperationCms,
                           Axis64Pos := "ManualOperationControl_U1Em7".axis,
                           AxisSoftCam := "ManualOperationControl_U1Em7".softCam,
                           twoWayAcutor := "ManualOperationControl_U1Em7".twoWayActuator,
                           Status := #StatusEm[7].Status,
                           errorID := #errorIDEm[7].errorID);
END_REGION

REGION Network 18 (SCL): Equipment Module 8 Cms Mapping
   REGION Input Mapping
        // Axis
       "ManualOperationControl_U1Em8".axis[1].monitoring := "Unit1.Em8.HmiInterface".cmThicknessAxisZ.monitoring;

       // SoftCam
       "ManualOperationControl_U1Em8".softCam[1] := "Unit1.Em8.HmiInterface".cm.softcam.thicknessAxisZ;

       // TwoWayActuator
       "ManualOperationControl_U1Em8".twoWayActuator[1].monitoring := "Unit1.Em8.HmiInterface".cmHipotTabContactorBwdFwd.monitoring;
       "ManualOperationControl_U1Em8".twoWayActuator[2].monitoring := "Unit1.Em8.HmiInterface".cmHipotTabContactorLeftOpenClose.monitoring;
       "ManualOperationControl_U1Em8".twoWayActuator[3].monitoring := "Unit1.Em8.HmiInterface".cmHipotTabContactorRightOpenClose.monitoring;
       "ManualOperationControl_U1Em8".twoWayActuator[6].monitoring := "Unit1.Em8.HmiInterface".cmHipotThicknessStageLiftFrontUpDown.monitoring;
       "ManualOperationControl_U1Em8".twoWayActuator[7].monitoring := "Unit1.Em8.HmiInterface".cmHipotThicknessStageLiftRearUpDown.monitoring;
   END_REGION


   REGION Output Mapping
       // Axis
       "Unit1.Em8.HmiInterface".cmThicknessAxisZ.commands.jogForward := "ManualOperationControl_U1Em8".axis[1].commands.jogForward;
       "Unit1.Em8.HmiInterface".cmThicknessAxisZ.commands.jogBackward := "ManualOperationControl_U1Em8".axis[1].commands.jogBackward;

       // TwoWayActuator
       "Unit1.Em8.HmiInterface".cmHipotTabContactorBwdFwd.commands := "ManualOperationControl_U1Em8".twoWayActuator[1].commands;
       "Unit1.Em8.HmiInterface".cmHipotTabContactorLeftOpenClose.commands := "ManualOperationControl_U1Em8".twoWayActuator[2].commands;
       "Unit1.Em8.HmiInterface".cmHipotTabContactorRightOpenClose.commands := "ManualOperationControl_U1Em8".twoWayActuator[3].commands;
       "Unit1.Em8.HmiInterface".cmHipotThicknessStageLiftFrontUpDown.commands := "ManualOperationControl_U1Em8".twoWayActuator[6].commands;
       "Unit1.Em8.HmiInterface".cmHipotThicknessStageLiftRearUpDown.commands := "ManualOperationControl_U1Em8".twoWayActuator[7].commands;
   END_REGION
END_REGION

REGION Network 19: Equipment Module 8
   RUNG wire#powerrail
      "CallManualOperationLines_EM"(disableUnit := #disableUnit1, manualOperationEm := "ManualOperationControl_U1Em8".manualOperationEm, manualOperationEmArea := "ManualOperationControl_U1Em8".manualOperationEmArea, manualOperationCms := "ManualOperationControl_U1Em8".manualOperationCms, Axis64Pos := "ManualOperationControl_U1Em8".axis, AxisSoftCam := "ManualOperationControl_U1Em8".softCam, twoWayAcutor := "ManualOperationControl_U1Em8".twoWayActuator, Status := #StatusEm[8].Status, errorID := #errorIDEm[8].errorID)
   END_RUNG
   // the same network as SCL:
   "CallManualOperationLines_EM"(disableUnit := #disableUnit1,
                           manualOperationEm := "ManualOperationControl_U1Em8".manualOperationEm,
                           manualOperationEmArea := "ManualOperationControl_U1Em8".manualOperationEmArea,
                           manualOperationCms := "ManualOperationControl_U1Em8".manualOperationCms,
                           Axis64Pos := "ManualOperationControl_U1Em8".axis,
                           AxisSoftCam := "ManualOperationControl_U1Em8".softCam,
                           twoWayAcutor := "ManualOperationControl_U1Em8".twoWayActuator,
                           Status := #StatusEm[8].Status,
                           errorID := #errorIDEm[8].errorID);
END_REGION

REGION Network 20 (SCL): Equipment Module 9 Cms Mapping
   REGION Input Mapping
       // TwoWayActuator
       "ManualOperationControl_U1Em9".twoWayActuator[1].monitoring := "Unit1.Em9.HmiInterface".cmVisionStageLiftUpDown.monitoring;
       "ManualOperationControl_U1Em9".twoWayActuator[2].monitoring := "Unit1.Em9.HmiInterface".cmVisionLightUpDown.monitoring;
   END_REGION


   REGION Output Mapping   
       // TwoWayActuator
       "Unit1.Em9.HmiInterface".cmVisionStageLiftUpDown.commands := "ManualOperationControl_U1Em9".twoWayActuator[1].commands;
       "Unit1.Em9.HmiInterface".cmVisionLightUpDown.commands := "ManualOperationControl_U1Em9".twoWayActuator[2].commands;
   END_REGION
END_REGION

REGION Network 21: Equipment Module 9
   RUNG wire#powerrail
      "CallManualOperationLines_EM"(disableUnit := #disableUnit1, manualOperationEm := "ManualOperationControl_U1Em9".manualOperationEm, manualOperationEmArea := "ManualOperationControl_U1Em9".manualOperationEmArea, manualOperationCms := "ManualOperationControl_U1Em9".manualOperationCms, Axis64Pos := "ManualOperationControl_U1Em9".axis, AxisSoftCam := "ManualOperationControl_U1Em9".softCam, twoWayAcutor := "ManualOperationControl_U1Em9".twoWayActuator, Status := #StatusEm[9].Status, errorID := #errorIDEm[9].errorID)
   END_RUNG
   // the same network as SCL:
   "CallManualOperationLines_EM"(disableUnit := #disableUnit1,
                           manualOperationEm := "ManualOperationControl_U1Em9".manualOperationEm,
                           manualOperationEmArea := "ManualOperationControl_U1Em9".manualOperationEmArea,
                           manualOperationCms := "ManualOperationControl_U1Em9".manualOperationCms,
                           Axis64Pos := "ManualOperationControl_U1Em9".axis,
                           AxisSoftCam := "ManualOperationControl_U1Em9".softCam,
                           twoWayAcutor := "ManualOperationControl_U1Em9".twoWayActuator,
                           Status := #StatusEm[9].Status,
                           errorID := #errorIDEm[9].errorID);
END_REGION

REGION Network 22 (SCL): Equipment Module 10 Cms Mapping
   REGION Input Mapping
       // TwoWayActuator
       "ManualOperationControl_U1Em10".twoWayActuator[1].monitoring := "Unit1.Em10.HmiInterface".cmLaserMarkCoverUpDown.monitoring;
       "ManualOperationControl_U1Em10".twoWayActuator[2].monitoring := "Unit1.Em10.HmiInterface".cmLaserMarkStageLiftUpDown.monitoring;
   END_REGION


   REGION Output Mapping 
       // TwoWayActuator
       "Unit1.Em10.HmiInterface".cmLaserMarkCoverUpDown.commands := "ManualOperationControl_U1Em10".twoWayActuator[1].commands;
       "Unit1.Em10.HmiInterface".cmLaserMarkStageLiftUpDown.commands := "ManualOperationControl_U1Em10".twoWayActuator[2].commands;
   END_REGION
END_REGION

REGION Network 23: Equipment Module 10
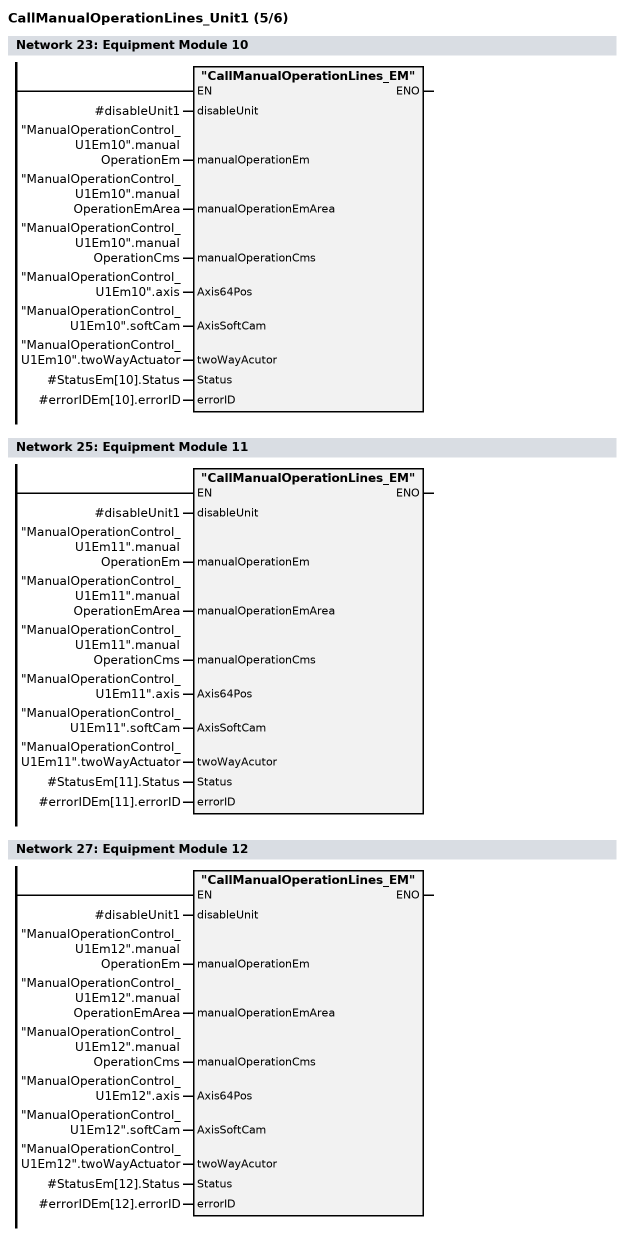
   RUNG wire#powerrail
      "CallManualOperationLines_EM"(disableUnit := #disableUnit1, manualOperationEm := "ManualOperationControl_U1Em10".manualOperationEm, manualOperationEmArea := "ManualOperationControl_U1Em10".manualOperationEmArea, manualOperationCms := "ManualOperationControl_U1Em10".manualOperationCms, Axis64Pos := "ManualOperationControl_U1Em10".axis, AxisSoftCam := "ManualOperationControl_U1Em10".softCam, twoWayAcutor := "ManualOperationControl_U1Em10".twoWayActuator, Status := #StatusEm[10].Status, errorID := #errorIDEm[10].errorID)
   END_RUNG
   // the same network as SCL:
   "CallManualOperationLines_EM"(disableUnit := #disableUnit1,
                           manualOperationEm := "ManualOperationControl_U1Em10".manualOperationEm,
                           manualOperationEmArea := "ManualOperationControl_U1Em10".manualOperationEmArea,
                           manualOperationCms := "ManualOperationControl_U1Em10".manualOperationCms,
                           Axis64Pos := "ManualOperationControl_U1Em10".axis,
                           AxisSoftCam := "ManualOperationControl_U1Em10".softCam,
                           twoWayAcutor := "ManualOperationControl_U1Em10".twoWayActuator,
                           Status := #StatusEm[10].Status,
                           errorID := #errorIDEm[10].errorID);
END_REGION

REGION Network 24 (SCL): Equipment Module 11 Cms Mapping
   REGION Input Mapping
       // TwoWayActuator
       "ManualOperationControl_U1Em11".twoWayActuator[1].monitoring := "Unit1.Em11.HmiInterface".cmWeightCheckStageLiftUpDown.monitoring;
   END_REGION


   REGION Output Mapping
       // TwoWayActuator
       "Unit1.Em11.HmiInterface".cmWeightCheckStageLiftUpDown.commands := "ManualOperationControl_U1Em11".twoWayActuator[1].commands;
   END_REGION
END_REGION

REGION Network 25: Equipment Module 11
   RUNG wire#powerrail
      "CallManualOperationLines_EM"(disableUnit := #disableUnit1, manualOperationEm := "ManualOperationControl_U1Em11".manualOperationEm, manualOperationEmArea := "ManualOperationControl_U1Em11".manualOperationEmArea, manualOperationCms := "ManualOperationControl_U1Em11".manualOperationCms, Axis64Pos := "ManualOperationControl_U1Em11".axis, AxisSoftCam := "ManualOperationControl_U1Em11".softCam, twoWayAcutor := "ManualOperationControl_U1Em11".twoWayActuator, Status := #StatusEm[11].Status, errorID := #errorIDEm[11].errorID)
   END_RUNG
   // the same network as SCL:
   "CallManualOperationLines_EM"(disableUnit := #disableUnit1,
                           manualOperationEm := "ManualOperationControl_U1Em11".manualOperationEm,
                           manualOperationEmArea := "ManualOperationControl_U1Em11".manualOperationEmArea,
                           manualOperationCms := "ManualOperationControl_U1Em11".manualOperationCms,
                           Axis64Pos := "ManualOperationControl_U1Em11".axis,
                           AxisSoftCam := "ManualOperationControl_U1Em11".softCam,
                           twoWayAcutor := "ManualOperationControl_U1Em11".twoWayActuator,
                           Status := #StatusEm[11].Status,
                           errorID := #errorIDEm[11].errorID);
END_REGION

REGION Network 26 (SCL): Equipment Module 12 Cms Mapping
   REGION Input Mapping
       // TwoWayActuator
       "ManualOperationControl_U1Em12".twoWayActuator[1].monitoring := "Unit1.Em12.HmiInterface".cmStackNgBoxClampMoverOpenClose.monitoring;
       "ManualOperationControl_U1Em12".twoWayActuator[2].monitoring := "Unit1.Em12.HmiInterface".cmStackNgBoxClampLeftOpenClose.monitoring;
       "ManualOperationControl_U1Em12".twoWayActuator[3].monitoring := "Unit1.Em12.HmiInterface".cmStackNgBoxClampRightOpenClose.monitoring;
       "ManualOperationControl_U1Em12".twoWayActuator[4].monitoring := "Unit1.Em12.HmiInterface".cmStackNgBoxLoadingUpDown.monitoring;
       "ManualOperationControl_U1Em12".twoWayActuator[5].monitoring := "Unit1.Em12.HmiInterface".cmStackNgBoxUnitMoverBwdFwd.monitoring;
       "ManualOperationControl_U1Em12".twoWayActuator[6].monitoring := "Unit1.Em12.HmiInterface".cmStackNgBoxLiftDownUp.monitoring;
       "ManualOperationControl_U1Em12".twoWayActuator[7].monitoring := "Unit1.Em12.HmiInterface".cmStackNgBoxLockDownUp.monitoring;
   END_REGION


   REGION Output Mapping
       // TwoWayActuator
       "Unit1.Em12.HmiInterface".cmStackNgBoxClampMoverOpenClose.commands := "ManualOperationControl_U1Em12".twoWayActuator[1].commands;
       "Unit1.Em12.HmiInterface".cmStackNgBoxClampLeftOpenClose.commands := "ManualOperationControl_U1Em12".twoWayActuator[2].commands;
       "Unit1.Em12.HmiInterface".cmStackNgBoxClampRightOpenClose.commands := "ManualOperationControl_U1Em12".twoWayActuator[3].commands;
       "Unit1.Em12.HmiInterface".cmStackNgBoxLoadingUpDown.commands := "ManualOperationControl_U1Em12".twoWayActuator[4].commands;
       "Unit1.Em12.HmiInterface".cmStackNgBoxUnitMoverBwdFwd.commands := "ManualOperationControl_U1Em12".twoWayActuator[5].commands;
       "Unit1.Em12.HmiInterface".cmStackNgBoxLiftDownUp.commands := "ManualOperationControl_U1Em12".twoWayActuator[6].commands;
       "Unit1.Em12.HmiInterface".cmStackNgBoxLockDownUp.commands := "ManualOperationControl_U1Em12".twoWayActuator[7].commands;
   END_REGION
END_REGION

REGION Network 27: Equipment Module 12
   RUNG wire#powerrail
      "CallManualOperationLines_EM"(disableUnit := #disableUnit1, manualOperationEm := "ManualOperationControl_U1Em12".manualOperationEm, manualOperationEmArea := "ManualOperationControl_U1Em12".manualOperationEmArea, manualOperationCms := "ManualOperationControl_U1Em12".manualOperationCms, Axis64Pos := "ManualOperationControl_U1Em12".axis, AxisSoftCam := "ManualOperationControl_U1Em12".softCam, twoWayAcutor := "ManualOperationControl_U1Em12".twoWayActuator, Status := #StatusEm[12].Status, errorID := #errorIDEm[12].errorID)
   END_RUNG
   // the same network as SCL:
   "CallManualOperationLines_EM"(disableUnit := #disableUnit1,
                           manualOperationEm := "ManualOperationControl_U1Em12".manualOperationEm,
                           manualOperationEmArea := "ManualOperationControl_U1Em12".manualOperationEmArea,
                           manualOperationCms := "ManualOperationControl_U1Em12".manualOperationCms,
                           Axis64Pos := "ManualOperationControl_U1Em12".axis,
                           AxisSoftCam := "ManualOperationControl_U1Em12".softCam,
                           twoWayAcutor := "ManualOperationControl_U1Em12".twoWayActuator,
                           Status := #StatusEm[12].Status,
                           errorID := #errorIDEm[12].errorID);
END_REGION

REGION Network 28 (SCL): Equipment Module 13 Cms Mapping
   REGION Input Mapping
        // Axis
       "ManualOperationControl_U1Em13".axis[1].monitoring := "Unit1.Em13.HmiInterface".cmJRUnloadingPnPAxisX.monitoring;
       "ManualOperationControl_U1Em13".axis[2].monitoring := "Unit1.Em13.HmiInterface".cmJRUnloadingPnPAxisZ.monitoring;
       "ManualOperationControl_U1Em13".axis[3].monitoring := "Unit1.Em13.HmiInterface".cmJRUnloadingPnPAxisC.monitoring;

       // SoftCam
       "ManualOperationControl_U1Em13".softCam[1] := "Unit1.Em13.HmiInterface".cm.softcam.jrUnIoadingPnPAxisX;
       "ManualOperationControl_U1Em13".softCam[2] := "Unit1.Em13.HmiInterface".cm.softcam.jrUnIoadingPnPAxisZ;
       "ManualOperationControl_U1Em13".softCam[3] := "Unit1.Em13.HmiInterface".cm.softcam.jrUnIoadingPnPAxisC;

       // TwoWayActuator
       "ManualOperationControl_U1Em13".twoWayActuator[1].monitoring := "Unit1.Em13.HmiInterface".cmJRUnloadingPnPClampOpenClose.monitoring;
   END_REGION


   REGION Output Mapping
       // Axis
       "Unit1.Em13.HmiInterface".cmJRUnloadingPnPAxisX.commands.jogForward := "ManualOperationControl_U1Em13".axis[1].commands.jogForward;
       "Unit1.Em13.HmiInterface".cmJRUnloadingPnPAxisX.commands.jogBackward := "ManualOperationControl_U1Em13".axis[1].commands.jogBackward;
       "Unit1.Em13.HmiInterface".cmJRUnloadingPnPAxisZ.commands.jogForward := "ManualOperationControl_U1Em13".axis[2].commands.jogForward;
       "Unit1.Em13.HmiInterface".cmJRUnloadingPnPAxisZ.commands.jogBackward := "ManualOperationControl_U1Em13".axis[2].commands.jogBackward;
       "Unit1.Em13.HmiInterface".cmJRUnloadingPnPAxisC.commands.jogForward := "ManualOperationControl_U1Em13".axis[3].commands.jogForward;
       "Unit1.Em13.HmiInterface".cmJRUnloadingPnPAxisC.commands.jogBackward := "ManualOperationControl_U1Em13".axis[3].commands.jogBackward;

       // TwoWayActuator
       "Unit1.Em13.HmiInterface".cmJRUnloadingPnPClampOpenClose.commands := "ManualOperationControl_U1Em13".twoWayActuator[1].commands;
   END_REGION
END_REGION

REGION Network 29: Equipment Module 13
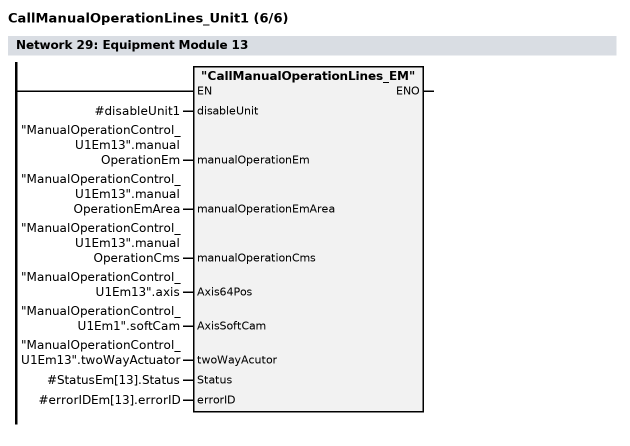
   RUNG wire#powerrail
      "CallManualOperationLines_EM"(disableUnit := #disableUnit1, manualOperationEm := "ManualOperationControl_U1Em13".manualOperationEm, manualOperationEmArea := "ManualOperationControl_U1Em13".manualOperationEmArea, manualOperationCms := "ManualOperationControl_U1Em13".manualOperationCms, Axis64Pos := "ManualOperationControl_U1Em13".axis, AxisSoftCam := "ManualOperationControl_U1Em1".softCam, twoWayAcutor := "ManualOperationControl_U1Em13".twoWayActuator, Status := #StatusEm[13].Status, errorID := #errorIDEm[13].errorID)
   END_RUNG
   // the same network as SCL:
   "CallManualOperationLines_EM"(disableUnit := #disableUnit1,
                           manualOperationEm := "ManualOperationControl_U1Em13".manualOperationEm,
                           manualOperationEmArea := "ManualOperationControl_U1Em13".manualOperationEmArea,
                           manualOperationCms := "ManualOperationControl_U1Em13".manualOperationCms,
                           Axis64Pos := "ManualOperationControl_U1Em13".axis,
                           AxisSoftCam := "ManualOperationControl_U1Em1".softCam,
                           twoWayAcutor := "ManualOperationControl_U1Em13".twoWayActuator,
                           Status := #StatusEm[13].Status,
                           errorID := #errorIDEm[13].errorID);
END_REGION
END_FUNCTION
